{attribute 'qualified_only'}
{attribute 'strict'}
TYPE eTest :
(
	enum_member := 0
);
END_TYPE

(* stored: Version 1.1.0.1, ProductVersion 3.1.4024.6
   DUT eTest: Id {e8534124-574b-4bad-b9ab-9f379405f450} *)
